FUNCTION_BLOCK OBDSS
  (* Standard: 61499-2 *)
  (* Version 0.1, 2015-00-24, Jin, Jin-PC *)
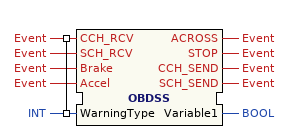
  EVENT_INPUT
    CCH_RCV WITH WarningType;
    SCH_RCV;
    Brake;
    Accel;
  END_EVENT
  EVENT_OUTPUT
    ACROSS;
    STOP;
    CCH_SEND;
    SCH_SEND;
  END_EVENT
  VAR_INPUT
    WarningType : INT;
  END_VAR
  VAR_OUTPUT
    Variable1 : BOOL;
  END_VAR
  ALGORITHM InputMultiplex IN C:

  END_ALGORITHM
END_FUNCTION_BLOCK
(* other elements stored in the file *)
(* ECC Name=OBDSS *)
(* ECState Name=WarningSystem *)
(* ECC Name=Brake *)
(* ECState Name=WaitBrake *)
(* ECState Name=BrakeWarning *)
(* ECAction Algorithm=InputMultiplex Output=CCH_SEND *)
(* ECTransition Source=WaitBrake Destination=BrakeWarning Condition=Brake *)
(* ECTransition Source=BrakeWarning Destination=BrakeWarning Condition=Brake *)
(* ECTransition Source=BrakeWarning Destination=WaitBrake Condition=true *)
(* ECC Name=Acceleration *)
(* ECState Name=WaitAccel *)
(* ECState Name=AccelWarning *)
(* ECAction Algorithm=InputMultiplex Output=CCH_SEND *)
(* ECTransition Source=WaitAccel Destination=AccelWarning Condition=Accel *)
(* ECTransition Source=AccelWarning Destination=AccelWarning Condition=Accel *)
(* ECTransition Source=AccelWarning Destination=WaitAccel Condition=true *)
(* ECC Name=TrafficLight *)
(* ECState Name=WaitLight *)
(* ECState Name=Across *)
(* ECAction Output=ACROSS *)
(* ECTransition Source=WaitLight Destination=Across Condition=CCH_RCV AND (WarningType = 1) *)
(* ECTransition Source=Across Destination=WaitLight Condition=true *)
(* ECC Name=Accidents *)
(* ECState Name=WaitEmergency *)
(* ECState Name=Stop *)
(* ECAction Output=STOP *)
(* ECTransition Source=WaitEmergency Destination=Stop Condition=CCH_RCV AND (WarningType = 0) *)
(* ECTransition Source=Stop Destination=WaitEmergency Condition=true *)
(* ECC Name=Region1 *)
(* ECState Name=State1 *)
(* ECState Name=State2 *)
(* ECTransition Source=State1 Destination=State1 Condition=true *)
(* ECTransition Source=State1 Destination=State2 Condition=true *)
